INTERFACE ITF_Component1_HMI_Connector_View EXTENDS ITF_BaseComponent_HMI_Connector_View

END_INTERFACE

(* stored: Version 1.1.0.1
   Itf ITF_Component1_HMI_Connector_View: Id {5cfd61a4-3b36-0372-1a6e-d9c24c09677f} *)
